Fanuc KAREL source: XML_SCAN.kl

PROGRAM T
%NOLOCKGROUP
VAR
 v0 : FILE
 v1 : STRING[40]
 v2 : INTEGER
 v3 : INTEGER
BEGIN
 XML_SCAN(v0, v1, v2, v3)
END T
